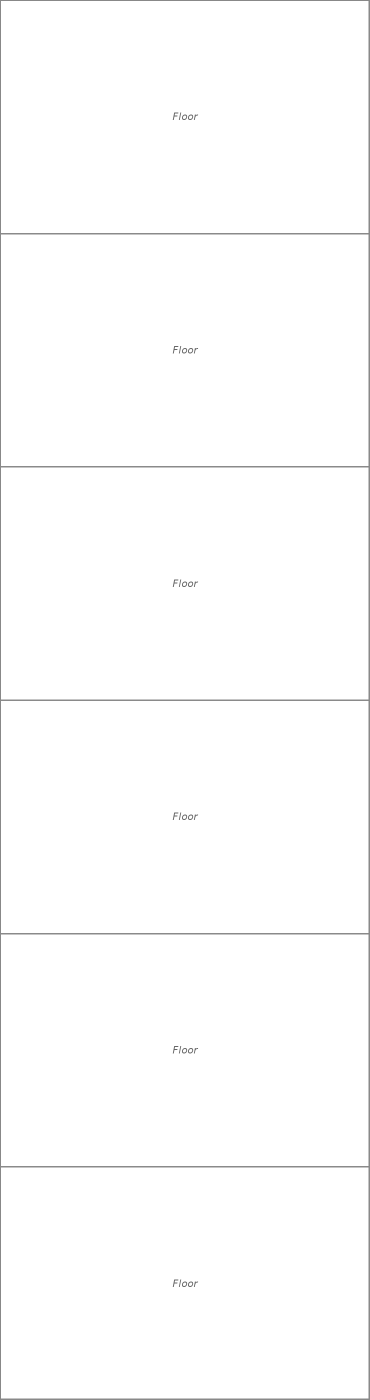
VISUALIZATION Lift_Floors  // 376x1422
VAR_IN_OUT
	Color 			: DWORD;
	Door_1_Position	: REAL;
	Door_1_M_Open	: BOOL;
	Door_1_M_Close	: BOOL;
	Door_2_Position	: REAL;
	
	Door_2_M_Open	: BOOL;
	Door_2_M_Close	: BOOL;
	Door_3_Position	: REAL;
	
	Door_3_M_Open	: BOOL;
	Door_3_M_Close	: BOOL;
	Door_4_Position	: REAL;
	
	Door_4_M_Open	: BOOL;
	Door_4_M_Close	: BOOL;
	Door_5_Position	: REAL;
	
	Door_5_M_Open	: BOOL;
	Door_5_M_Close	: BOOL;
	Door_6_Position	: REAL;
	
	Door_6_M_Open	: BOOL;
	Door_6_M_Close	: BOOL;
	
	LED_Up_1 		: BOOL;
	LED_Down_1 		: BOOL;
	FloorNumber_1 	: INT;
	BtnLed_1 		: ARRAY[1..6] OF BOOL;;
	Btn_1			: ARRAY[1..6] OF BOOL;
	LB_1 			: BOOL;
	LED_DoorOpen_1 	: BOOL;
	LED_DoorClosed_1: BOOL;

	LED_Up_2 		: BOOL;
	LED_Down_2 		: BOOL;
	FloorNumber_2 	: INT;
	BtnLed_2 		: ARRAY[1..6] OF BOOL;;
	Btn_2			: ARRAY[1..6] OF BOOL;
	LB_2 			: BOOL;
	LED_DoorOpen_2 	: BOOL;
	LED_DoorClosed_2: BOOL;


	LED_Up_3 		: BOOL;
	LED_Down_3 		: BOOL;
	FloorNumber_3 	: INT;
	BtnLed_3 		: ARRAY[1..6] OF BOOL;;
	Btn_3			: ARRAY[1..6] OF BOOL;
	LB_3 			: BOOL;
	LED_DoorOpen_3 	: BOOL;
	LED_DoorClosed_3: BOOL;

	LED_Up_4 		: BOOL;
	LED_Down_4 		: BOOL;
	FloorNumber_4 	: INT;
	BtnLed_4 		: ARRAY[1..6] OF BOOL;;
	Btn_4			: ARRAY[1..6] OF BOOL;
	LB_4 			: BOOL;
	LED_DoorOpen_4 	: BOOL;
	LED_DoorClosed_4: BOOL;

	LED_Up_5 		: BOOL;
	LED_Down_5 		: BOOL;
	FloorNumber_5 	: INT;
	BtnLed_5 		: ARRAY[1..6] OF BOOL;;
	Btn_5			: ARRAY[1..6] OF BOOL;
	LB_5 			: BOOL;
	LED_DoorOpen_5 	: BOOL;
	LED_DoorClosed_5: BOOL;

	LED_Up_6 		: BOOL;
	LED_Down_6 		: BOOL;
	FloorNumber_6 	: INT;
	BtnLed_6 		: ARRAY[1..6] OF BOOL;;
	Btn_6			: ARRAY[1..6] OF BOOL;
	LB_6 			: BOOL;
	LED_DoorOpen_6 	: BOOL;
	LED_DoorClosed_6: BOOL;

END_VAR
    Frame (0,1185 376x237)
        shows Floor(Color := Color, LED_Up := LED_Up_1, LED_Down := LED_Down_1, FloorNumber := FloorNumber_1, BtnLed := BtnLed_1, Btn := Btn_1, LB := LB_1, LED_DoorOpen := LED_DoorOpen_1, LED_DoorClosed := LED_DoorClosed_1, PositionDoor := Door_1_Position, M_Open := Door_1_M_Open, M_Close := Door_1_M_Close)
    Frame (0,948 376x237)
        shows Floor(Color := Color, LED_Up := LED_Up_2, LED_Down := LED_Down_2, FloorNumber := FloorNumber_2, BtnLed := BtnLed_2, Btn := Btn_2, LB := LB_2, LED_DoorOpen := LED_DoorOpen_2, LED_DoorClosed := LED_DoorClosed_2, PositionDoor := Door_2_Position, M_Open := Door_2_M_Open, M_Close := Door_2_M_Close)
    Frame (0,711 376x237)
        shows Floor(Color := Color, LED_Up := LED_Up_3, LED_Down := LED_Down_3, FloorNumber := FloorNumber_3, BtnLed := BtnLed_3, Btn := Btn_3, LB := LB_3, LED_DoorOpen := LED_DoorOpen_3, LED_DoorClosed := LED_DoorClosed_3, PositionDoor := Door_3_Position, M_Open := Door_3_M_Open, M_Close := Door_3_M_Close)
    Frame (0,474 376x237)
        shows Floor(Color := Color, LED_Up := LED_Up_4, LED_Down := LED_Down_4, FloorNumber := FloorNumber_4, BtnLed := BtnLed_4, Btn := Btn_4, LB := LB_4, LED_DoorOpen := LED_DoorOpen_4, LED_DoorClosed := LED_DoorClosed_4, PositionDoor := Door_4_Position, M_Open := Door_4_M_Open, M_Close := Door_4_M_Close)
    Frame (0,237 376x237)
        shows Floor(Color := Color, LED_Up := LED_Up_5, LED_Down := LED_Down_5, FloorNumber := FloorNumber_5, BtnLed := BtnLed_5, Btn := Btn_5, LB := LB_5, LED_DoorOpen := LED_DoorOpen_5, LED_DoorClosed := LED_DoorClosed_5, PositionDoor := Door_5_Position, M_Open := Door_5_M_Open, M_Close := Door_5_M_Close)
    Frame (0,0 376x237)
        shows Floor(Color := Color, LED_Up := LED_Up_6, LED_Down := LED_Down_6, FloorNumber := FloorNumber_6, BtnLed := BtnLed_6, Btn := Btn_6, LB := LB_6, LED_DoorOpen := LED_DoorOpen_6, LED_DoorClosed := LED_DoorClosed_6, PositionDoor := Door_6_Position, M_Open := Door_6_M_Open, M_Close := Door_6_M_Close)
END_VISUALIZATION

(* stored: Version 1.1.0.1
   Visu Lift_Floors: Id {d4667ef1-e109-462c-aad2-e1caf1fdd3d4} *)
